{attribute addProperty BoxType "EK1100-0000-0018"}
{attribute addProperty Id "Beckhoff_EL37xxEK1122Beckhoff_EL37xxEK1122_36723BB4162A_0001_EL3702_0000_0002EL3702_72DB3B7943454.25A_0002_EL3702_0000_0003EL3702_72DB3B7943454.25A_0003_EL3702_0015_0003EL3702_72DB3B7943454.25A_0004_EL3742_0000_0001EL3742_56C06C6414818.5A_0005_EL3742_0000_0002EL3742_72DB3B7943454.25A_0006_EL3742_0000_0003EL3742_72DB3B7943454.25A_0007_EL3751_0000_0020EL3751_1042CC8027434.25A_0008_EL3751_0000_0021EL3751_1042CC8027434.25A_0009_EL3751_0000_0022EL3751_1042CC8027434.25A_0010_EL3751_0000_0023EL3751_1042CC8027434.25A_0011_EL3751_0004_0022EL3751_1042CC8027434.25A_0012_EL3751_0004_0023EL3751_1042CC8027434.25A_0013_EL3751_0020_0020EL3751_1042CC8027434.25A_0014_EL3751_0020_0021EL3751_1042CC8027434.25A_0015_EL3751_0020_0022EL3751_1042CC8027434.25A_0016_EL3751_0020_0023EL3751_1042CC8027434.25A_0017_EL3751_0024_0022EL3751_1042CC8027434.25A_0018_EL3751_0024_0023EL3751_1042CC8027434.25A_0019_EL3773_0000_0016EL3773_90A9FC821282160.25A_0020_EL3773_0000_0017EL3773_C057E1551282160.25A_0021_EL3773_0000_0018EL3773_D6945B001282160.25A_0022_EL3773_0000_0019EL3773_40CB6C261282160.25A_0023_EL3773_0000_0020EL3773_40CB6C261282160.25A_0024_EL3773_0000_0021EL3773_40CB6C261282160.25A_0025_EL3783_0000_0018EL3783_81B4F6712282285.25"}
{attribute addProperty CRC "1935173602"}
{attribute addProperty SizeInBites "15596"}
{attribute addProperty SizeInBytes "1949.5"}
TYPE Beckhoff_EL37xx_735867E2 EXTENDS EK1100_179A0949 :
STRUCT
	{attribute addProperty Name "Beckhoff_EL37xxEK1122"}
	Beckhoff_EL37xxEK1122 : Beckhoff_EL37xxEK1122_36723BB4;
	{attribute addProperty Name "A_0001_EL3702_0000_0002"}
	A_0001_EL3702_0000_0002 : EL3702_72DB3B79;
	{attribute addProperty Name "A_0002_EL3702_0000_0003"}
	A_0002_EL3702_0000_0003 : EL3702_72DB3B79;
	{attribute addProperty Name "A_0003_EL3702_0015_0003"}
	A_0003_EL3702_0015_0003 : EL3702_72DB3B79;
	{attribute addProperty Name "A_0004_EL3742_0000_0001"}
	A_0004_EL3742_0000_0001 : EL3742_56C06C64;
	{attribute addProperty Name "A_0005_EL3742_0000_0002"}
	A_0005_EL3742_0000_0002 : EL3742_72DB3B79;
	{attribute addProperty Name "A_0006_EL3742_0000_0003"}
	A_0006_EL3742_0000_0003 : EL3742_72DB3B79;
	{attribute addProperty Name "A_0007_EL3751_0000_0020"}
	A_0007_EL3751_0000_0020 : EL3751_1042CC80;
	{attribute addProperty Name "A_0008_EL3751_0000_0021"}
	A_0008_EL3751_0000_0021 : EL3751_1042CC80;
	{attribute addProperty Name "A_0009_EL3751_0000_0022"}
	A_0009_EL3751_0000_0022 : EL3751_1042CC80;
	{attribute addProperty Name "A_0010_EL3751_0000_0023"}
	A_0010_EL3751_0000_0023 : EL3751_1042CC80;
	{attribute addProperty Name "A_0011_EL3751_0004_0022"}
	A_0011_EL3751_0004_0022 : EL3751_1042CC80;
	{attribute addProperty Name "A_0012_EL3751_0004_0023"}
	A_0012_EL3751_0004_0023 : EL3751_1042CC80;
	{attribute addProperty Name "A_0013_EL3751_0020_0020"}
	A_0013_EL3751_0020_0020 : EL3751_1042CC80;
	{attribute addProperty Name "A_0014_EL3751_0020_0021"}
	A_0014_EL3751_0020_0021 : EL3751_1042CC80;
	{attribute addProperty Name "A_0015_EL3751_0020_0022"}
	A_0015_EL3751_0020_0022 : EL3751_1042CC80;
	{attribute addProperty Name "A_0016_EL3751_0020_0023"}
	A_0016_EL3751_0020_0023 : EL3751_1042CC80;
	{attribute addProperty Name "A_0017_EL3751_0024_0022"}
	A_0017_EL3751_0024_0022 : EL3751_1042CC80;
	{attribute addProperty Name "A_0018_EL3751_0024_0023"}
	A_0018_EL3751_0024_0023 : EL3751_1042CC80;
	{attribute addProperty Name "A_0019_EL3773_0000_0016"}
	A_0019_EL3773_0000_0016 : EL3773_90A9FC82;
	{attribute addProperty Name "A_0020_EL3773_0000_0017"}
	A_0020_EL3773_0000_0017 : EL3773_C057E155;
	{attribute addProperty Name "A_0021_EL3773_0000_0018"}
	A_0021_EL3773_0000_0018 : EL3773_D6945B00;
	{attribute addProperty Name "A_0022_EL3773_0000_0019"}
	A_0022_EL3773_0000_0019 : EL3773_40CB6C26;
	{attribute addProperty Name "A_0023_EL3773_0000_0020"}
	A_0023_EL3773_0000_0020 : EL3773_40CB6C26;
	{attribute addProperty Name "A_0024_EL3773_0000_0021"}
	A_0024_EL3773_0000_0021 : EL3773_40CB6C26;
	{attribute addProperty Name "A_0025_EL3783_0000_0018"}
	A_0025_EL3783_0000_0018 : EL3783_81B4F671;
END_STRUCT
END_TYPE

(* stored: Version 1.2.0.0, ProductVersion 3.1.4024.9
   DUT Beckhoff_EL37xx_735867E2: Id {9b674387-db72-4a7b-ada0-e7c95cc19ddf} *)
